PROGRAM PRG_TEST
VAR
	fbCheckPartTest		: FB_CellCheckPart_Test;
END_VAR

TcUnit.RUN();

END_PROGRAM

(* stored: Version 1.1.0.1, ProductVersion 3.1.4024.12
   POU PRG_TEST: Id {d8ef3780-da63-4f67-b013-b5f69f0f0425}, SpecialFunc None *)
